Yaskawa INFORM job: X2SCHODKI_ZEW.JBI

/JOB
//NAME X2SCHODKI_ZEW
//POS
///NPOS 223,223,223,10,0,0
///TOOL 0
///POSTYPE PULSE
///PULSE
C00000=21160,-126487,-99095,6220,53097,19917
C00001=122314,-84956,-84267,5758,65294,20346
C00002=113867,-2788,-32259,11364,77586,-20622
C00003=111699,9606,-11794,12514,71800,-21939
C00004=110873,16102,-4909,12893,71047,-22311
C00005=111426,18220,-2948,12689,70847,-22135
C00006=111334,17863,-3281,12723,70881,-22164
C00007=111334,17842,-1921,12786,70054,-22254
C00008=111688,13758,-7042,12574,71029,-22022
C00009=137921,23655,2193,-26065,80546,13065
C00010=138187,30095,8478,-26164,80127,13260
C00011=137141,31636,10013,-25924,79665,12972
C00012=137283,31426,9804,-25956,79727,13011
C00013=137283,31447,11085,-26011,79025,13166
C00014=137811,24810,3269,-26040,80453,13045
C00015=130093,15204,-5597,-17076,73087,3422
C00016=130254,16762,-4164,-17139,73044,3486
C00017=130499,11823,-8660,-17205,73314,3535
C00018=136657,16032,-4835,-19303,74485,5576
C00019=136779,34044,12201,-19450,73350,5806
C00020=136367,37287,16065,-19383,72578,5782
C00021=135529,38270,17077,-19116,72272,5524
C00022=135735,38345,17156,-19186,72312,5593
C00023=135735,38391,18179,-19247,71738,5687
C00024=136093,38073,17157,-19317,72259,5733
C00025=136821,38987,18103,-19565,72324,5991
C00026=137234,41236,20445,-19732,72152,6174
C00027=137468,37941,16529,-19737,72884,6137
C00028=139273,33119,8814,-10616,74138,14432
C00029=138400,39162,15428,-10360,73077,14220
C00030=137624,40756,17090,-10099,72782,13973
C00031=137810,40443,16764,-10163,72844,14033
C00032=137810,40460,18419,-10216,71849,14119
C00033=138377,33107,10032,-10341,73283,14197
C00034=129933,32626,9546,1459,71562,3103
C00035=130107,34413,11352,1398,71367,3162
C00036=130344,28976,5916,1305,71915,3250
C00037=134876,30968,7890,-396,71698,4822
C00038=142592,70732,50995,-12851,68399,16892
C00039=141830,71409,51797,-12602,68137,16639
C00040=142006,70894,51186,-12652,68274,16689
C00041=142006,71149,52557,-12712,67578,16765
C00042=142006,71007,51815,-12679,67954,16725
C00043=142747,76515,58410,-13043,66871,17119
C00044=142702,66110,44987,-12780,69711,16790
C00045=130401,22900,-3912,9781,74013,14096
C00046=130750,-77898,-76934,10038,67211,13654
C00047=128341,-94500,-64478,15665,37561,8814
C00048=125354,-34494,-33676,16070,41961,8103
C00049=123908,-22688,-35224,-7311,60763,8117
C00050=115329,1774,-22996,-8583,68206,33205
C00051=113811,6923,-16554,-7934,66753,32769
C00052=112938,8598,-15088,-7517,66630,32466
C00053=113357,7607,-15958,-7718,66694,32611
C00054=113357,7474,-14642,-7767,65823,32669
C00055=113357,7562,-15559,-7732,66427,32629
C00056=114674,8046,-17033,-9196,71995,10105
C00057=114277,9137,-16073,-9034,71921,9973
C00058=114994,10710,-14679,-9331,71949,10219
C00059=115929,5782,-19714,-10610,72890,11247
C00060=114914,9168,-18033,-20160,83408,25507
C00061=114509,10465,-16323,-20060,82947,25443
C00062=114509,10278,-15209,-20089,82211,25564
C00063=114509,10430,-16126,-20066,82816,25464
C00064=113574,12027,-14696,-19812,82540,25184
C00065=113966,9476,-16971,-19916,82715,25292
C00066=109195,41890,2270,-19889,88323,22522
C00067=109420,41611,2136,-14547,83651,24420
C00068=109633,43097,3705,-14621,83493,24508
C00069=110073,47498,8361,-9922,80898,20177
C00070=110340,48514,8983,-10012,81065,20250
C00071=109875,50139,10594,-6927,80049,17487
C00072=111642,41129,-2073,-7513,83338,17864
C00073=120740,-4591,-30289,-15267,55452,23675
C00074=120758,-111403,-89341,-20679,37744,27189
C00075=120758,-111403,-89341,-20679,37744,27189
C00076=97140,-41370,-74515,11864,90116,-15742
C00077=93918,-16818,-51601,15265,90472,-19448
C00078=96838,-21310,-54909,14446,89719,-18600
C00079=97144,-22320,-55662,14359,89616,-18514
C00080=98771,-24881,-57497,13895,89173,-18041
C00081=115828,-29996,-61044,-7286,86100,2495
C00082=121364,-24267,-57094,-13933,89260,9154
C00083=125066,-13537,-49221,-14991,90516,10198
C00084=125405,-12324,-48437,-15087,90711,10281
C00085=127775,-3453,-41245,-15747,91251,10973
C00086=117906,-11103,-47413,-1372,86513,-3179
C00087=107817,-4833,-42392,13913,90158,-17947
C00088=111065,-8601,-45456,12965,89620,-16971
C00089=111228,-9142,-45834,12917,89553,-16926
C00090=113235,-11504,-47787,12324,89257,-16321
C00091=116129,-16038,-53218,11461,89860,-15351
C00092=132129,3503,-37461,731,88042,-5165
C00093=134839,10104,-29765,-1476,86561,-3078
C00094=133535,10494,-29542,-1044,86604,-3481
C00095=133472,10527,-29512,-1023,86602,-3500
C00096=132997,13157,-27039,-5636,86965,851
C00097=131112,-12606,-50888,-7793,88905,29033
C00098=129834,-10958,-47906,-7386,87816,28703
C00099=133351,1378,-37957,-8503,88347,29764
C00100=133639,2898,-36665,-8594,88358,29852
C00101=132895,14544,-26435,-2898,86896,24452
C00102=133144,15405,-25686,-2979,86883,24528
C00103=133588,9909,-35564,-3125,90148,24585
C00104=114600,-38617,-66572,24501,76796,21744
C00105=88804,-102668,-113384,34072,81784,13502
C00106=-3643,-76224,-106676,-19950,71810,-76872
C00107=-6047,-95755,-92046,14751,98253,-9605
C00108=-2299,-70459,-84112,3705,91093,-18065
C00109=-2299,-70459,-84112,3705,91093,-18065
C00110=-2299,-70459,-84112,3705,91093,-18065
C00111=-2299,-70459,-84112,3705,91093,-18065
C00112=61951,-108908,-90353,7974,21769,-53190
C00113=44975,-75191,-76287,54105,62461,-71292
C00114=78581,-58710,-61930,31634,35162,-55381
C00115=94816,-22771,-39143,38147,43253,-85351
C00116=95668,-20492,-32997,40754,37729,-87628
C00117=95668,-20442,-31356,41600,36978,-88107
C00118=95668,-20481,-32513,41001,37505,-87770
C00119=95495,-18068,-30743,41020,37699,-87770
C00120=95668,-20481,-32513,41001,37505,-87770
C00121=89708,-21268,-34265,45191,40885,-89740
C00122=90261,-15540,-28471,45297,40161,-89843
C00123=90261,-15513,-27582,45749,39780,-90110
C00124=90261,-15527,-28007,45532,39961,-89983
C00125=91375,-15045,-27644,44668,39419,-89560
C00126=90261,-15527,-28007,45532,39961,-89983
C00127=88067,4046,-12693,46606,41526,-90451
C00128=88067,4066,-11724,47089,41117,-90741
C00129=88067,4053,-12277,46812,41349,-90575
C00130=89178,4455,-11933,46018,40776,-90188
C00131=88067,4046,-12908,46498,41617,-90387
C00132=93864,-1171,-17172,27469,32670,-81316
C00133=93864,-1150,-16127,27931,32107,-81561
C00134=93864,-1161,-16600,27720,32361,-81450
C00135=93686,724,-15030,27925,32421,-81546
C00136=93864,-1171,-17458,27343,32827,-81250
C00137=86880,-2670,-19039,34652,35541,-84684
C00138=77447,40941,12142,46518,66528,-79108
C00139=77447,40828,13235,46743,66015,-79371
C00140=77447,40915,12396,46570,66408,-79170
C00141=78189,41279,12776,46293,66002,-79003
C00142=77447,40915,12396,46570,66408,-79170
C00143=77711,61383,34518,44784,60703,-78470
C00144=77711,61401,35861,45103,60114,-78770
C00145=77711,61383,34367,44748,60769,-78437
C00146=78627,62334,35456,44423,60182,-78251
C00147=77711,61383,34367,44748,60769,-78437
C00148=87327,38488,-37,11684,57539,-57739
C00149=92703,33891,441,-7168,52274,-42102
C00150=94252,42993,11540,-8600,52099,-41498
C00151=94252,42798,12742,-8697,51267,-41425
C00152=94252,42977,11640,-8607,52029,-41490
C00153=94205,45159,13958,-8608,51725,-41483
C00154=94252,42977,11640,-8607,52029,-41490
C00155=88553,40317,7447,-4237,52798,-43866
C00156=77780,64504,35767,30085,55551,-63063
C00157=77882,64751,36053,30043,55472,-63041
C00158=77882,64734,37138,30274,54883,-63228
C00159=77882,64751,36157,30064,55416,-63059
C00160=78504,65403,36908,29747,55085,-62879
C00161=77882,64751,36157,30064,55416,-63059
C00162=77930,65478,35918,25842,53172,-64425
C00163=75957,78225,52136,32216,53612,-64557
C00164=75957,78336,53316,32477,53042,-64758
C00165=75957,78231,52217,32233,53572,-64572
C00166=76543,78457,52489,31920,53306,-64380
C00167=75957,78231,52217,32233,53572,-64572
C00168=75783,52857,14963,26033,68951,-61065
C00169=76778,51540,16645,25850,67104,-61119
C00170=76553,54259,19675,26040,66751,-61289
C00171=76152,68337,35819,26754,64443,-62008
C00172=76309,68979,36633,26729,64087,-61973
C00173=76161,73805,46213,28343,55084,-61966
C00174=76040,75497,47702,28425,55082,-62022
C00175=75485,77195,52229,31394,50715,-63899
C00176=76358,61277,29656,23751,52989,-59172
C00177=75244,23807,-9833,23130,57943,-58480
C00178=78328,30150,-3634,21247,56637,-57509
C00179=82524,40429,3879,10756,62616,-55403
C00180=83243,40821,5102,10290,61963,-55146
C00181=92066,29463,-1741,-9440,53850,-44784
C00182=92409,29931,-1279,-9693,53846,-44645
C00183=95822,30058,-1154,-12140,54276,-43316
C00184=92072,29548,-1666,-1163,53131,-49252
C00185=90114,17633,-16179,284,55928,-50028
C00186=80680,14818,-24193,20442,65844,-59872
C00187=77180,38928,7111,43331,74666,-71993
C00188=76673,54469,24090,43953,73098,-72919
C00189=76771,55672,25429,43962,72900,-72963
C00190=76784,55849,25626,43964,72871,-72969
C00191=78172,63512,34338,39520,65661,-69940
C00192=79648,59091,29288,35397,62522,-67074
C00193=75980,37060,-454,35377,69732,-66149
C00194=81483,21043,-13915,32107,67437,-64274
C00195=93507,15990,-19907,5211,64480,-50669
C00196=99800,11020,-22513,-5623,60000,-50039
C00197=99783,5101,-23986,-5176,53212,-49502
C00198=100096,6075,-23185,433,53012,-52451
C00199=100559,6099,-23054,81,52942,-52266
C00200=100559,6099,-23054,81,52942,-52266
C00201=95780,-7481,-38206,3595,55393,-54089
C00202=86068,-7258,-38029,32714,65078,-69570
C00203=89977,-5445,-32844,31222,61873,-68759
C00204=89643,-3500,-31211,31407,61985,-68864
C00205=88246,9256,-20330,32202,62368,-69333
C00206=88278,10099,-19644,32183,62365,-69319
C00207=87437,19709,-10754,32777,62224,-69720
C00208=93562,10508,-19170,18010,55559,-61503
C00209=91617,5056,-25544,19093,57043,-62018
C00210=90732,-18366,-45622,16723,54511,-62954
C00211=99990,-18392,-38429,13920,44377,-71620
C00212=100890,-18558,-38626,13099,44267,-71210
C00213=97938,-19656,-35927,25966,40954,-77255
C00214=98057,-22963,-34084,32871,34362,-85156
C00215=99570,-14469,-34407,26946,45535,-82523
C00216=93873,-14551,-28302,47146,43784,-90863
C00217=93873,-14551,-28302,47146,43784,-90863
C00218=92894,-25654,-38538,40707,40207,-87648
C00219=51114,-81290,-74278,61960,52593,-60278
C00220=6076,-109546,-85200,71251,79672,-70600
C00221=6076,-109546,-85200,71251,79672,-70600
C00222=6076,-109546,-85200,-4239,76823,-70600
BC00000=277643,516186,172088
BC00001=328181,496789,172088
BC00002=328180,496788,172085
BC00003=328180,496788,172085
BC00004=328180,496788,172085
BC00005=328180,496788,172085
BC00006=328180,496788,172085
BC00007=328180,496788,172085
BC00008=328180,496788,172085
BC00009=328180,496788,172085
BC00010=328180,496788,172085
BC00011=328180,496788,172085
BC00012=328180,496788,172085
BC00013=328180,496788,172085
BC00014=328180,496788,172085
BC00015=328180,496788,172085
BC00016=328180,496788,172085
BC00017=328180,496788,172085
BC00018=328180,496788,172085
BC00019=328180,496788,172085
BC00020=328180,496788,172085
BC00021=328180,496788,172085
BC00022=328180,496788,172085
BC00023=328180,496788,172085
BC00024=328180,496788,172085
BC00025=328180,496788,172085
BC00026=328180,496788,172085
BC00027=328180,496788,172085
BC00028=328180,496788,172085
BC00029=328180,496788,172085
BC00030=328180,496788,172085
BC00031=328180,496788,172085
BC00032=328180,496788,172085
BC00033=328180,496788,172085
BC00034=328180,496788,172085
BC00035=328180,496788,172085
BC00036=328180,496788,172085
BC00037=328180,496788,172085
BC00038=328180,496788,172085
BC00039=328180,496788,172085
BC00040=328180,496788,172085
BC00041=328180,496788,172085
BC00042=328180,496788,172085
BC00043=328180,496788,172085
BC00044=328180,496788,172085
BC00045=328180,496788,172085
BC00046=328180,496788,172085
BC00047=194416,502028,172085
BC00048=194416,502028,172085
BC00049=173311,425006,172085
BC00050=173311,425006,140819
BC00051=173311,425006,140819
BC00052=173311,425006,140819
BC00053=173311,425006,140819
BC00054=173311,425006,140819
BC00055=173311,425006,140819
BC00056=173311,425006,140819
BC00057=173311,425006,140819
BC00058=173311,425006,140819
BC00059=173311,425006,140819
BC00060=173311,425006,140819
BC00061=173311,425006,140819
BC00062=173311,425006,140819
BC00063=173311,425006,140819
BC00064=173311,425006,140819
BC00065=173311,425006,140819
BC00066=158492,452266,59327
BC00067=158492,452266,59327
BC00068=158492,452266,59327
BC00069=158492,452266,59327
BC00070=158492,452266,59327
BC00071=158492,452266,59327
BC00072=158492,452266,59327
BC00073=158492,452266,59327
BC00074=158492,507957,59327
BC00075=293306,507957,59327
BC00076=293305,437676,59324
BC00077=293305,437676,59324
BC00078=293305,437676,59324
BC00079=293305,437676,59324
BC00080=293305,437676,59324
BC00081=293305,437676,59324
BC00082=293305,437676,59324
BC00083=293305,437676,59324
BC00084=293305,437676,59324
BC00085=293305,437676,59324
BC00086=293305,437676,59324
BC00087=293305,437676,59324
BC00088=293305,437676,59324
BC00089=293305,437676,59324
BC00090=293305,437676,59324
BC00091=293305,437676,59324
BC00092=293305,437676,59324
BC00093=293305,437676,59324
BC00094=293305,437676,59324
BC00095=293305,437676,59324
BC00096=293305,437676,59324
BC00097=293305,437676,59324
BC00098=293305,437676,59324
BC00099=293305,437676,59324
BC00100=293305,437676,59324
BC00101=293305,437676,59324
BC00102=293305,437676,59324
BC00103=293305,437676,59324
BC00104=293305,437676,59324
BC00105=293305,491548,59324
BC00106=199448,515539,1075137
BC00107=95028,515070,919110
BC00108=123826,515279,972180
BC00109=123826,515279,972180
BC00110=123826,515279,972180
BC00111=44761,462630,27794
BC00112=44761,462630,27794
BC00113=44761,462630,27793
BC00114=44761,462630,27793
BC00115=44761,462630,27793
BC00116=44761,462631,27793
BC00117=44761,462631,27793
BC00118=44761,462631,27793
BC00119=44761,462631,27793
BC00120=44761,462631,27793
BC00121=44761,462631,27793
BC00122=44761,462631,27793
BC00123=44761,462631,27793
BC00124=44761,462631,27793
BC00125=44761,462631,27793
BC00126=44761,462631,27793
BC00127=44761,462631,27793
BC00128=44761,462631,27793
BC00129=44761,462631,27793
BC00130=44761,462631,27793
BC00131=44761,462631,27793
BC00132=44761,462631,27793
BC00133=44761,462631,27793
BC00134=44761,462631,27793
BC00135=44761,462631,27793
BC00136=44761,462631,27793
BC00137=44761,462631,27793
BC00138=44761,462631,27793
BC00139=44761,462631,27793
BC00140=44761,462631,27793
BC00141=44761,462631,27793
BC00142=44761,462631,27793
BC00143=44761,462631,27793
BC00144=44761,462631,27793
BC00145=44761,462631,27793
BC00146=44761,462631,27793
BC00147=44761,462631,27793
BC00148=44761,462631,27793
BC00149=44761,462630,27793
BC00150=44761,462630,27793
BC00151=44761,462630,27793
BC00152=44761,462630,27793
BC00153=44761,462630,27793
BC00154=44761,462630,27793
BC00155=44761,462630,27793
BC00156=44761,462630,27793
BC00157=44761,462630,27793
BC00158=44761,462630,27793
BC00159=44761,462630,27793
BC00160=44761,462630,27793
BC00161=44761,462630,27793
BC00162=44761,453221,27793
BC00163=44761,453221,27793
BC00164=44761,453221,27793
BC00165=44761,453221,27793
BC00166=44761,453221,27793
BC00167=44761,453221,27793
BC00168=45255,444613,27793
BC00169=45255,444613,27793
BC00170=45255,444613,27793
BC00171=45255,444613,27793
BC00172=45255,444613,27793
BC00173=45255,444613,27793
BC00174=45255,444613,27793
BC00175=45255,444613,27793
BC00176=45255,444613,27793
BC00177=45255,444613,27793
BC00178=45255,444613,27793
BC00179=45255,444613,27793
BC00180=45253,444683,27793
BC00181=45253,444683,27793
BC00182=45253,444683,27793
BC00183=45253,444683,27793
BC00184=45253,444683,27793
BC00185=45253,444683,27793
BC00186=44971,454975,27792
BC00187=44971,454975,27792
BC00188=44971,454975,27792
BC00189=44971,454975,27792
BC00190=44971,454975,27792
BC00191=44970,454994,27792
BC00192=44970,454994,27792
BC00193=44970,454994,27792
BC00194=44966,455154,27792
BC00195=44966,455154,27792
BC00196=44966,455154,27792
BC00197=44966,455154,27792
BC00198=44966,455154,27792
BC00199=44966,455154,27792
BC00200=44966,455154,27792
BC00201=44966,455154,27792
BC00202=44966,455154,27792
BC00203=44957,455470,27792
BC00204=44957,455470,27792
BC00205=44957,455470,27792
BC00206=44957,455470,27792
BC00207=44957,455470,27792
BC00208=44957,455470,27792
BC00209=44957,455470,27792
BC00210=44859,459040,27792
BC00211=44823,460358,27792
BC00212=44823,460358,27792
BC00213=44823,460358,27792
BC00214=44823,460358,27792
BC00215=44823,460358,27792
BC00216=44823,460358,27792
BC00217=44823,460358,27792
BC00218=44823,460358,27792
BC00219=44761,462630,27793
BC00220=44761,546100,27793
BC00221=44761,546100,27793
BC00222=44761,546100,971290
EC00000=798156,-183832
EC00001=798156,-183832
EC00002=798153,-183831
EC00003=798153,-183831
EC00004=798153,-183831
EC00005=798153,-183831
EC00006=798153,-183831
EC00007=798153,-183831
EC00008=798153,-183831
EC00009=798153,-183831
EC00010=798153,-183831
EC00011=798153,-183831
EC00012=798153,-183831
EC00013=798153,-183831
EC00014=798153,-183831
EC00015=798153,-183831
EC00016=798153,-183831
EC00017=798153,-183831
EC00018=798153,-183831
EC00019=798153,-183831
EC00020=798153,-183831
EC00021=798153,-183831
EC00022=798153,-183831
EC00023=798153,-183831
EC00024=798153,-183831
EC00025=798153,-183831
EC00026=798153,-183831
EC00027=798153,-183831
EC00028=798153,-183831
EC00029=798153,-183831
EC00030=798153,-183831
EC00031=798153,-183831
EC00032=798153,-183831
EC00033=798153,-183831
EC00034=798153,-183831
EC00035=798153,-183831
EC00036=798153,-183831
EC00037=798153,-183831
EC00038=798153,-183831
EC00039=798153,-183831
EC00040=798153,-183831
EC00041=798153,-183831
EC00042=798153,-183831
EC00043=798153,-183831
EC00044=798153,-183831
EC00045=798153,-183831
EC00046=798153,-183831
EC00047=798153,-183831
EC00048=798153,-183831
EC00049=798153,-183831
EC00050=798153,-183831
EC00051=798153,-183831
EC00052=798153,-183831
EC00053=798153,-183831
EC00054=798153,-183831
EC00055=798153,-183831
EC00056=798153,-183831
EC00057=798153,-183831
EC00058=798153,-183831
EC00059=798153,-183831
EC00060=798153,-183831
EC00061=798153,-183831
EC00062=798153,-183831
EC00063=798153,-183831
EC00064=798153,-183831
EC00065=798153,-183831
EC00066=798153,-183831
EC00067=798153,-183831
EC00068=798153,-183831
EC00069=798153,-183831
EC00070=798153,-183831
EC00071=798153,-183831
EC00072=798153,-183831
EC00073=798153,-183831
EC00074=798153,-183831
EC00075=798153,-183831
EC00076=798151,-183830
EC00077=798151,-183830
EC00078=798151,-183830
EC00079=798151,-183830
EC00080=798151,-183830
EC00081=798151,-183830
EC00082=798151,-183830
EC00083=798151,-183830
EC00084=798151,-183830
EC00085=798151,-183830
EC00086=798151,-183830
EC00087=798151,-183830
EC00088=798151,-183830
EC00089=798151,-183830
EC00090=798151,-183830
EC00091=798151,-183830
EC00092=798151,-183830
EC00093=798151,-183830
EC00094=798151,-183830
EC00095=798151,-183830
EC00096=798151,-183830
EC00097=798151,-183830
EC00098=798151,-183830
EC00099=798151,-183830
EC00100=798151,-183830
EC00101=798151,-183830
EC00102=798151,-183830
EC00103=798151,-183830
EC00104=798151,-183830
EC00105=798151,-183830
EC00106=798151,-183830
EC00107=798156,-183832
EC00108=322978,-183832
EC00109=357094,925242
EC00110=800604,925242
EC00111=800604,925242
EC00112=800604,925242
EC00113=800603,925242
EC00114=800603,925242
EC00115=800603,925242
EC00116=800600,925239
EC00117=800600,925239
EC00118=800600,925239
EC00119=800600,925239
EC00120=800600,925239
EC00121=800600,925239
EC00122=800600,925239
EC00123=800600,925239
EC00124=800600,925239
EC00125=800600,925239
EC00126=800600,925239
EC00127=800600,925239
EC00128=800600,925239
EC00129=800600,925239
EC00130=800600,925239
EC00131=800600,925239
EC00132=800600,925239
EC00133=800600,925239
EC00134=800600,925239
EC00135=800600,925239
EC00136=800600,925239
EC00137=800600,925239
EC00138=800600,925239
EC00139=800600,925239
EC00140=800600,925239
EC00141=800600,925239
EC00142=800600,925239
EC00143=800600,925239
EC00144=800600,925239
EC00145=800600,925239
EC00146=800600,925239
EC00147=800600,925239
EC00148=800600,925239
EC00149=800600,925239
EC00150=800600,925239
EC00151=800600,925239
EC00152=800600,925239
EC00153=800600,925239
EC00154=800600,925239
EC00155=800600,925239
EC00156=800600,925239
EC00157=800600,925239
EC00158=800600,925239
EC00159=800600,925239
EC00160=800600,925239
EC00161=800600,925239
EC00162=800600,925239
EC00163=800600,925239
EC00164=800600,925239
EC00165=800600,925239
EC00166=800600,925239
EC00167=800600,925239
EC00168=800600,925239
EC00169=800600,925239
EC00170=800600,925239
EC00171=800600,925239
EC00172=800600,925239
EC00173=800600,925239
EC00174=800600,925239
EC00175=800600,925239
EC00176=800600,925239
EC00177=800600,925239
EC00178=800600,925239
EC00179=800600,925239
EC00180=800600,925239
EC00181=800600,925239
EC00182=800600,925239
EC00183=800600,925239
EC00184=800600,925239
EC00185=800600,925239
EC00186=800598,925237
EC00187=800598,925237
EC00188=800598,925237
EC00189=800598,925237
EC00190=800598,925237
EC00191=800598,925237
EC00192=800598,925237
EC00193=800598,925237
EC00194=800598,925237
EC00195=800598,925237
EC00196=800598,925237
EC00197=800598,925237
EC00198=800598,925237
EC00199=800598,925237
EC00200=800598,925237
EC00201=800598,925237
EC00202=800598,925237
EC00203=800598,925237
EC00204=800598,925237
EC00205=800598,925237
EC00206=800598,925237
EC00207=800598,925237
EC00208=800598,925237
EC00209=800598,925237
EC00210=800598,925237
EC00211=800600,925239
EC00212=800600,925239
EC00213=800600,925239
EC00214=800600,925239
EC00215=800600,925239
EC00216=800600,925239
EC00217=800600,925239
EC00218=800600,925239
EC00219=800603,925242
EC00220=800603,925242
EC00221=-11362,925242
EC00222=-11362,925242
///POSTYPE BASE
///RECTAN
///RCONF 0,0,0,0,1,0,0,0,0,0,0,0,0,0,0,0,0,0,0,0,0,0,0,0
P00006=2.006,1.622,-0.565,0.0000,0.0000,0.0000
P00021=0.073,2.058,-0.109,0.0000,0.0000,0.0000
P00022=2.006,1.622,-0.565,0.0000,0.0000,0.0000
///RCONF 0,0,0,0,0,0,0,0,0,0,0,0,0,0,0,0,0,0,0,0,0,0,0,0
P00023=-2.957,-4.083,2.762,0.0000,0.0000,0.0000
P00024=-1.466,-0.226,-0.419,0.0000,0.0000,0.0000
P00025=3.643,0.007,-2.585,0.0000,0.0000,0.0000
P00026=2.644,0.055,-2.583,0.0000,0.0000,0.0000
P00027=2.278,0.099,-4.210,0.0000,0.0000,0.0000
P00028=-1.778,-0.182,-2.050,0.0000,0.0000,0.0000
P00029=1.749,4.006,-0.261,0.0000,0.0000,0.0000
//INST
///DATE 2024/12/16 21:22
///ATTR SC,RW
///GROUP1 RB1,BS1
///GROUP2 ST1
NOP
MOVJ C00000 BC00000 VJ=100.00  +MOVJ EC00000 VJ=100.00
MOVJ C00001 BC00001 VJ=100.00  +MOVJ EC00001 VJ=100.00
MOVJ C00002 BC00002 VJ=100.00  +MOVJ EC00002 VJ=100.00
SMOVL C00003 BC00003 V=833.3  +MOVJ EC00003
SMOVL C00004 BC00004 V=166.7  +MOVJ EC00004
SREFP 3 C00005 BC00005  +REFP EC00005
CALL JOB:SEARCH-R1-S13D
SET P021 P006
SFTON3D P021
SMOVL C00006 BC00006 V=166.7  +MOVJ EC00006
SREFP 3 C00007 BC00007  +REFP EC00007
CALL JOB:SEARCH-R1-S13D
SET P021 P006
SFTON3D P021
SMOVL C00008 BC00008 V=166.7  +MOVJ EC00008
SFTOF3D
SMOVL C00009 BC00009 V=833.3  +MOVJ EC00009
SMOVL C00010 BC00010 V=166.7  +MOVJ EC00010
SREFP 3 C00011 BC00011  +REFP EC00011
CALL JOB:SEARCH-R1-S13D
SET P022 P006
SFTON3D P022
SMOVL C00012 BC00012 V=166.7  +MOVJ EC00012
SREFP 3 C00013 BC00013  +REFP EC00013
CALL JOB:SEARCH-R1-S13D
SET P022 P006
SFTON3D P022
SMOVL C00014 BC00014 V=166.7  +MOVJ EC00014
SMOVL C00015 BC00015 V=166.7  +MOVJ EC00015
SREFP 3 C00016 BC00016  +REFP EC00016
CALL JOB:SEARCH-R1-S13D
SET P022 P006
SFTON3D P022
SMOVL C00017 BC00017 V=166.7  +MOVJ EC00017
SFTOF3D
SMOVL C00018 BC00018 V=500.0  +MOVJ EC00018
SMOVL C00019 BC00019 V=500.0  +MOVJ EC00019
SMOVL C00020 BC00020 V=166.7  +MOVJ EC00020
SREFP 3 C00021 BC00021  +REFP EC00021
CALL JOB:SEARCH-R1-S13D
SET P023 P006
SFTON3D P023
SMOVL C00022 BC00022 V=166.7  +MOVJ EC00022
SREFP 3 C00023 BC00023  +REFP EC00023
CALL JOB:SEARCH-R1-S13D
SET P023 P006
SFTON3D P023
SMOVL C00024 BC00024 V=166.7  +MOVJ EC00024
SMOVL C00025 BC00025 V=166.7  +MOVJ EC00025
SREFP 3 C00026 BC00026  +REFP EC00026
CALL JOB:SEARCH-R1-S13D
SET P023 P006
SFTON3D P023
SMOVL C00027 BC00027 V=166.7  +MOVJ EC00027
SFTOF3D
SMOVL C00028 BC00028 V=333.3  +MOVJ EC00028
SMOVL C00029 BC00029 V=166.7  +MOVJ EC00029
SREFP 3 C00030 BC00030  +REFP EC00030
CALL JOB:SEARCH-R1-S13D
SET P024 P006
SFTON3D P024
SMOVL C00031 BC00031 V=166.7  +MOVJ EC00031
SREFP 3 C00032 BC00032  +REFP EC00032
CALL JOB:SEARCH-R1-S13D
SET P024 P006
SFTON3D P024
SMOVL C00033 BC00033 V=166.7  +MOVJ EC00033
SMOVL C00034 BC00034 V=166.7  +MOVJ EC00034
SREFP 3 C00035 BC00035  +REFP EC00035
CALL JOB:SEARCH-R1-S13D
SET P024 P006
SFTON3D P024
SMOVL C00036 BC00036 V=166.7  +MOVJ EC00036
SFTOF3D
SMOVL C00037 BC00037 V=333.3  +MOVJ EC00037
SMOVL C00038 BC00038 V=166.7  +MOVJ EC00038
SREFP 3 C00039 BC00039  +REFP EC00039
CALL JOB:SEARCH-R1-S13D
SET P025 P006
SFTON3D P025
SMOVL C00040 BC00040 V=166.7  +MOVJ EC00040
SREFP 3 C00041 BC00041  +REFP EC00041
CALL JOB:SEARCH-R1-S13D
SET P025 P006
SFTON3D P025
SMOVL C00042 BC00042 V=166.7  +MOVJ EC00042
SREFP 3 C00043 BC00043  +REFP EC00043
CALL JOB:SEARCH-R1-S13D
SET P025 P006
SFTON3D P025
SMOVL C00044 BC00044 V=166.7  +MOVJ EC00044
SFTOF3D
SMOVL C00045 BC00045 V=333.3  +MOVJ EC00045
SMOVL C00046 BC00046 V=1000.0  +MOVJ EC00046
SMOVL C00047 BC00047 V=1000.0  +MOVJ EC00047
SMOVL C00048 BC00048 V=1000.0  +MOVJ EC00048
SMOVL C00049 BC00049 V=666.7  +MOVJ EC00049
SMOVL C00050 BC00050 V=666.7  +MOVJ EC00050
SMOVL C00051 BC00051 V=166.7  +MOVJ EC00051
SREFP 3 C00052 BC00052  +REFP EC00052
CALL JOB:SEARCH-R1-S13D
SET P027 P006
SFTON3D P027
SMOVL C00053 BC00053 V=166.7  +MOVJ EC00053
SREFP 3 C00054 BC00054  +REFP EC00054
CALL JOB:SEARCH-R1-S13D
SET P027 P006
SFTON3D P027
SMOVL C00055 BC00055 V=166.7  +MOVJ EC00055
SMOVL C00056 BC00056 V=250.0  +MOVJ EC00056
SMOVL C00057 BC00057 V=250.0  +MOVJ EC00057
SREFP 3 C00058 BC00058  +REFP EC00058
CALL JOB:SEARCH-R1-S13D
SET P027 P006
SFTON3D P027
SMOVL C00059 BC00059 V=166.7  +MOVJ EC00059
SFTOF3D
SMOVL C00060 BC00060 V=250.0  +MOVJ EC00060
SMOVL C00061 BC00061 V=166.7  +MOVJ EC00061
SREFP 3 C00062 BC00062  +REFP EC00062
CALL JOB:SEARCH-R1-S13D
SET P026 P006
SFTON3D P026
SMOVL C00063 BC00063 V=166.7  +MOVJ EC00063
SREFP 3 C00064 BC00064  +REFP EC00064
CALL JOB:SEARCH-R1-S13D
SET P026 P006
SFTON3D P026
SMOVL C00065 BC00065 V=166.7  +MOVJ EC00065
MACRO1 MJ#(0) ARGF9
SMOVL C00066 BC00066 V=250.0  +MOVJ EC00066
ARCON
SMOVL C00067 BC00067 V=10.0  +MOVJ EC00067
SMOVL C00068 BC00068 V=10.0  +MOVJ EC00068
SFTON3D P027
SMOVL C00069 BC00069 V=10.0  +MOVJ EC00069
ARCOF
SMOVL C00070 BC00070 V=10.0  +MOVJ EC00070
ARCON
SMOVL C00071 BC00071 V=10.0  +MOVJ EC00071
ARCOF
SFTOF3D
SMOVL C00072 BC00072 V=250.0  +MOVJ EC00072
SMOVL C00073 BC00073 V=666.7  +MOVJ EC00073
SMOVL C00074 BC00074 V=666.7  +MOVJ EC00074
SMOVL C00075 BC00075 V=1000.0  +MOVJ EC00075
SMOVL C00076 BC00076 V=1000.0  +MOVJ EC00076
SFTON3D P021
SMOVL C00077 BC00077 V=166.7  +MOVJ EC00077
ARCON
SMOVL C00078 BC00078 V=10.0  +MOVJ EC00078
SFTON3D P022
SMOVL C00079 BC00079 V=10.0  +MOVJ EC00079
SMOVL C00080 BC00080 V=10.0  +MOVJ EC00080
SMOVL C00081 BC00081 V=10.0  +MOVJ EC00081
SMOVL C00082 BC00082 V=10.0  +MOVJ EC00082
SMOVL C00083 BC00083 V=10.0  +MOVJ EC00083
SMOVL C00084 BC00084 V=10.0  +MOVJ EC00084
SFTON3D P023
SMOVL C00085 BC00085 V=10.0  +MOVJ EC00085
SMOVL C00086 BC00086 V=10.0  +MOVJ EC00086
SMOVL C00087 BC00087 V=10.0  +MOVJ EC00087
SMOVL C00088 BC00088 V=10.0  +MOVJ EC00088
SFTON3D P024
SMOVL C00089 BC00089 V=10.0  +MOVJ EC00089
SMOVL C00090 BC00090 V=10.0  +MOVJ EC00090
ARCOF
SFTOF3D
SMOVL C00091 BC00091 V=250.0  +MOVJ EC00091
SMOVL C00092 BC00092 V=500.0  +MOVJ EC00092
SFTON3D P026
SMOVL C00093 BC00093 V=250.0  +MOVJ EC00093
ARCON
SMOVL C00094 BC00094 V=10.0  +MOVJ EC00094
SMOVL C00095 BC00095 V=10.0  +MOVJ EC00095
SFTON3D P025
SMOVL C00096 BC00096 V=10.0  +MOVJ EC00096
ARCOF
SFTOF3D
SMOVL C00097 BC00097 V=400.0  +MOVJ EC00097
SFTON3D P024
SMOVL C00098 BC00098 V=166.7  +MOVJ EC00098
ARCON
SMOVL C00099 BC00099 V=10.0  +MOVJ EC00099
SMOVL C00100 BC00100 V=10.0  +MOVJ EC00100
SFTON3D P025
SMOVL C00101 BC00101 V=10.0  +MOVJ EC00101
SMOVL C00102 BC00102 V=10.0  +MOVJ EC00102
ARCOF
SFTOF3D
SMOVL C00103 BC00103 V=250.0  +MOVJ EC00103
SMOVL C00104 BC00104 V=833.3  +MOVJ EC00104
MOVJ C00105 BC00105 VJ=100.00  +MOVJ EC00105 VJ=100.00
MOVJ C00106 BC00106 VJ=100.00  +MOVJ EC00106 VJ=100.00
CALL JOB:CLEAN-R1_KM_NEW
MOVJ C00107 BC00107 VJ=100.00  +MOVJ EC00107 VJ=100.00
PAUSE
MOVJ C00108 BC00108 VJ=100.00  +MOVJ EC00108 VJ=100.00
MOVJ C00109 BC00109 VJ=100.00  +MOVJ EC00109 VJ=100.00
MOVJ C00110 BC00110 VJ=100.00  +MOVJ EC00110 VJ=100.00
MOVJ C00111 BC00111 VJ=100.00  +MOVJ EC00111 VJ=100.00
MOVJ C00112 BC00112 VJ=100.00  +MOVJ EC00112 VJ=100.00
MOVJ C00113 BC00113 VJ=30.00  +MOVJ EC00113 VJ=100.00
MOVL C00114 BC00114 V=333.3  +MOVJ EC00114 VJ=30.00
MOVL C00115 BC00115 V=333.3  +MOVJ EC00115 VJ=30.00
SFTOF3D
SMOVL C00116 BC00116 V=166.7  +MOVJ EC00116
SREFP 3 C00117 BC00117  +REFP EC00117
CALL JOB:SEARCH-R1-S13D
SET P027 P006
SFTON3D P027
SMOVL C00118 BC00118 V=166.7  +MOVJ EC00118
SREFP 3 C00119 BC00119  +REFP EC00119
CALL JOB:SEARCH-R1-S13D
SET P027 P006
SFTON3D P027
SMOVL C00120 BC00120 V=166.7  +MOVJ EC00120
SFTOF3D
MOVL C00121 BC00121 V=333.3  +MOVJ EC00121 VJ=30.00
SFTOF3D
SMOVL C00122 BC00122 V=166.7  +MOVJ EC00122
SREFP 3 C00123 BC00123  +REFP EC00123
CALL JOB:SEARCH-R1-S13D
SET P026 P006
SFTON3D P026
SMOVL C00124 BC00124 V=166.7  +MOVJ EC00124
SREFP 3 C00125 BC00125  +REFP EC00125
CALL JOB:SEARCH-R1-S13D
SET P026 P006
SFTON3D P026
SMOVL C00126 BC00126 V=166.7  +MOVJ EC00126
SFTOF3D
SMOVL C00127 BC00127 V=166.7  +MOVJ EC00127
SREFP 3 C00128 BC00128  +REFP EC00128
CALL JOB:SEARCH-R1-S13D
SET P025 P006
SFTON3D P025
SMOVL C00129 BC00129 V=166.7  +MOVJ EC00129
SREFP 3 C00130 BC00130  +REFP EC00130
CALL JOB:SEARCH-R1-S13D
SET P025 P006
SFTON3D P025
SMOVL C00131 BC00131 V=166.7  +MOVJ EC00131
SFTOF3D
SMOVL C00132 BC00132 V=166.7  +MOVJ EC00132
SREFP 3 C00133 BC00133  +REFP EC00133
CALL JOB:SEARCH-R1-S13D
SET P024 P006
SFTON3D P024
SMOVL C00134 BC00134 V=166.7  +MOVJ EC00134
SREFP 3 C00135 BC00135  +REFP EC00135
CALL JOB:SEARCH-R1-S13D
SET P024 P006
SFTON3D P024
SMOVL C00136 BC00136 V=166.7  +MOVJ EC00136
SFTOF3D
MOVL C00137 BC00137 V=333.3  +MOVJ EC00137 VJ=30.00
SMOVL C00138 BC00138 V=166.7  +MOVJ EC00138
SREFP 3 C00139 BC00139  +REFP EC00139
CALL JOB:SEARCH-R1-S13D
SET P028 P006
SFTON3D P028
SMOVL C00140 BC00140 V=166.7  +MOVJ EC00140
SREFP 3 C00141 BC00141  +REFP EC00141
CALL JOB:SEARCH-R1-S13D
SET P028 P006
SFTON3D P028
SMOVL C00142 BC00142 V=166.7  +MOVJ EC00142
SFTOF3D
SMOVL C00143 BC00143 V=166.7  +MOVJ EC00143
SREFP 3 C00144 BC00144  +REFP EC00144
CALL JOB:SEARCH-R1-S13D
SET P023 P006
SFTON3D P023
SMOVL C00145 BC00145 V=166.7  +MOVJ EC00145
SREFP 3 C00146 BC00146  +REFP EC00146
CALL JOB:SEARCH-R1-S13D
SET P023 P006
SFTON3D P023
SMOVL C00147 BC00147 V=166.7  +MOVJ EC00147
SFTOF3D
MOVJ C00148 BC00148 VJ=50.00  +MOVJ EC00148 VJ=50.00
MOVJ C00149 BC00149 VJ=30.00  +MOVJ EC00149 VJ=30.00
SMOVL C00150 BC00150 V=166.7  +MOVJ EC00150
SREFP 3 C00151 BC00151  +REFP EC00151
CALL JOB:SEARCH-R1-S13D
SET P029 P006
SFTON3D P029
SMOVL C00152 BC00152 V=166.7  +MOVJ EC00152
SREFP 3 C00153 BC00153  +REFP EC00153
CALL JOB:SEARCH-R1-S13D
SET P029 P006
SFTON3D P029
SMOVL C00154 BC00154 V=166.7  +MOVJ EC00154
SFTOF3D
MOVL C00155 BC00155 V=333.3  +MOVJ EC00155 VJ=30.00
MOVL C00156 BC00156 V=333.3  +MOVJ EC00156 VJ=30.00
SMOVL C00157 BC00157 V=166.7  +MOVJ EC00157
SREFP 3 C00158 BC00158  +REFP EC00158
CALL JOB:SEARCH-R1-S13D
SET P022 P006
SFTON3D P022
SMOVL C00159 BC00159 V=166.7  +MOVJ EC00159
SREFP 3 C00160 BC00160  +REFP EC00160
CALL JOB:SEARCH-R1-S13D
SET P022 P006
SFTON3D P022
SMOVL C00161 BC00161 V=166.7  +MOVJ EC00161
SFTOF3D
MOVL C00162 BC00162 V=333.3  +MOVJ EC00162 VJ=30.00
SMOVL C00163 BC00163 V=166.7  +MOVJ EC00163
SREFP 3 C00164 BC00164  +REFP EC00164
CALL JOB:SEARCH-R1-S13D
SET P021 P006
SFTON3D P021
SMOVL C00165 BC00165 V=166.7  +MOVJ EC00165
SREFP 3 C00166 BC00166  +REFP EC00166
CALL JOB:SEARCH-R1-S13D
SET P021 P006
SFTON3D P021
SMOVL C00167 BC00167 V=166.7  +MOVJ EC00167
SMOVL C00168 BC00168 V=166.7  +MOVJ EC00168
MACRO1 MJ#(0) ARGF9
SFTON3D P022
SMOVL C00169 BC00169 V=166.7  +MOVJ EC00169
ARCON
SMOVL C00170 BC00170 V=10.0  +MOVJ EC00170
SMOVL C00171 BC00171 V=10.0  +MOVJ EC00171
SFTON3D P021
SMOVL C00172 BC00172 V=10.0  +MOVJ EC00172
SMOVL C00173 BC00173 V=10.0  +MOVJ EC00173
SMOVL C00174 BC00174 V=10.0  +MOVJ EC00174
SMOVL C00175 BC00175 V=10.0  +MOVJ EC00175
ARCOF
SFTOF3D
SMOVL C00176 BC00176 V=250.0  +MOVJ EC00176
SMOVL C00177 BC00177 V=250.0  +MOVJ EC00177
MOVJ C00178 BC00178 VJ=30.00  +MOVJ EC00178 VJ=30.00
SMOVL C00179 BC00179 V=250.0  +MOVJ EC00179
SFTON3D P029
SMOVL C00180 BC00180 V=250.0  +MOVJ EC00180
ARCON
SMOVL C00181 BC00181 V=10.0  +MOVJ EC00181
SMOVL C00182 BC00182 V=10.0  +MOVJ EC00182
SMOVL C00183 BC00183 V=10.0  +MOVJ EC00183
SMOVL C00184 BC00184 V=10.0  +MOVJ EC00184
ARCOF
SFTOF3D
SMOVL C00185 BC00185 V=333.3  +MOVJ EC00185
SMOVL C00186 BC00186 V=333.3  +MOVJ EC00186
SFTON3D P028
SMOVL C00187 BC00187 V=250.0  +MOVJ EC00187
ARCON
SMOVL C00188 BC00188 V=10.0  +MOVJ EC00188
SMOVL C00189 BC00189 V=10.0  +MOVJ EC00189
SMOVL C00190 BC00190 V=10.0  +MOVJ EC00190
SFTON3D P023
SMOVL C00191 BC00191 V=10.0  +MOVJ EC00191
SMOVL C00192 BC00192 V=10.0  +MOVJ EC00192
ARCOF
SFTOF3D
SMOVL C00193 BC00193 V=333.3  +MOVJ EC00193
SMOVL C00194 BC00194 V=333.3  +MOVJ EC00194
SFTON3D P024
SMOVL C00195 BC00195 V=166.7  +MOVJ EC00195
ARCON
SMOVL C00196 BC00196 V=10.0  +MOVJ EC00196
SMOVL C00197 BC00197 V=10.0  +MOVJ EC00197
SMOVL C00198 BC00198 V=10.0  +MOVJ EC00198
SMOVL C00199 BC00199 V=10.0  +MOVJ EC00199
SMOVL C00200 BC00200 V=10.0  +MOVJ EC00200
ARCOF
SFTOF3D
SMOVL C00201 BC00201 V=250.0  +MOVJ EC00201
SMOVL C00202 BC00202 V=250.0  +MOVJ EC00202
SFTON3D P026
SMOVL C00203 BC00203 V=250.0  +MOVJ EC00203
ARCON
SMOVL C00204 BC00204 V=10.0  +MOVJ EC00204
SMOVL C00205 BC00205 V=10.0  +MOVJ EC00205
SFTON3D P025
SMOVL C00206 BC00206 V=10.0  +MOVJ EC00206
SMOVL C00207 BC00207 V=10.0  +MOVJ EC00207
SMOVL C00208 BC00208 V=10.0  +MOVJ EC00208
ARCOF
SFTOF3D
SMOVL C00209 BC00209 V=250.0  +MOVJ EC00209
SMOVL C00210 BC00210 V=250.0  +MOVJ EC00210
SFTON3D P027
SMOVL C00211 BC00211 V=250.0  +MOVJ EC00211
ARCON
SMOVL C00212 BC00212 V=10.0  +MOVJ EC00212
SMOVL C00213 BC00213 V=10.0  +MOVJ EC00213
SMOVL C00214 BC00214 V=10.0  +MOVJ EC00214
SMOVL C00215 BC00215 V=10.0  +MOVJ EC00215
SMOVL C00216 BC00216 V=10.0  +MOVJ EC00216
SMOVL C00217 BC00217 V=10.0  +MOVJ EC00217
ARCOF
SFTOF3D
SMOVL C00218 BC00218 V=250.0  +MOVJ EC00218
SMOVL C00219 BC00219 V=250.0  +MOVJ EC00219
MOVJ C00220 BC00220 VJ=30.00  +MOVJ EC00220 VJ=30.00
MOVJ C00221 BC00221 VJ=100.00  +MOVJ EC00221 VJ=100.00
MOVJ C00222 BC00222 VJ=100.00  +MOVJ EC00222 VJ=100.00
END
